(* Logix 5000 project; controller Industrial Emulate 5570 rev 30.12; software revision 30.01 *)

TASK MainTask (continuous, watchdog 500 ms) : MainProgram

MODULES
   Local : Emulate 5570 (ICP 3, rev 30.12)
       : 1756-IB16 (ICP 0, rev 3.1, Input RPI 20 ms)
       : vendor 1 type 7 code 8 (ICP 1, rev 3.1, Output RPI 20 ms)
END_MODULES

PROGRAM MainProgram   (* main routine MainRoutine *)
VAR
   Close_PB : BOOL;
   Fully_close : ALIAS FOR Local:0:I.Data.3;
   Fully_open : ALIAS FOR Local:0:I.Data.1;
   Gate_close : ALIAS FOR Local:1:O.Data.1;
   Gate_Open : ALIAS FOR Local:1:O.Data.0;
   Green_light_indicate : BOOL;
   Prox_entrance_gate : ALIAS FOR Local:0:I.Data.2;
   prox_path_gate : ALIAS FOR Local:0:I.Data.0;
   Red_light_indicate : BOOL;
   Start_PB : BOOL;
   Timer_delay : TIMER := (PRE := 3000);
END_VAR

ROUTINE Controller   (* ladder *)
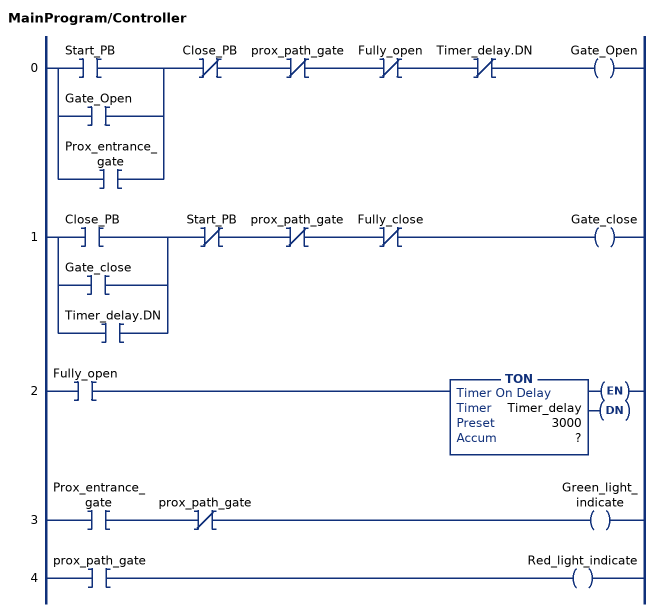
   0: [XIC(Start_PB) ,XIC(Gate_Open) ,XIC(Prox_entrance_gate) ]XIO(Close_PB)XIO(prox_path_gate)XIO(Fully_open)XIO(Timer_delay.DN)OTE(Gate_Open);
   1: [XIC(Close_PB) ,XIC(Gate_close) ,XIC(Timer_delay.DN) ]XIO(Start_PB)XIO(prox_path_gate)XIO(Fully_close)OTE(Gate_close);
   2: XIC(Fully_open)TON(Timer_delay,?,?);
   3: XIC(Prox_entrance_gate)XIO(prox_path_gate)OTE(Green_light_indicate);
   4: XIC(prox_path_gate)OTE(Red_light_indicate);
END_ROUTINE

ROUTINE MainRoutine   (* ladder *)
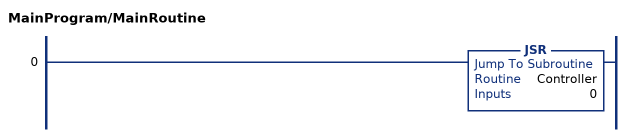
   0: JSR(Controller,0);
END_ROUTINE
END_PROGRAM
